// TIA Portal V17 export
// export: Created 2024-09-02T12:49:59.2213188Z, ExportSetting WithDefaults, DisplayName Totally Integrated Automation Portal, DisplayVersion V17, DisplayName TIA Portal Openness, DisplayVersion V17, DisplayName TIA Portal Version Control Interface, DisplayVersion V17, DisplayName STEP 7 Professional, DisplayVersion V17, DisplayName STEP 7 Safety, DisplayVersion V17, DisplayName WinCC Professional, DisplayVersion V17
DATA_BLOCK "LTLL_Data"   // DB556
TITLE = LTLL_Data
{ S7_Optimized_Access := 'TRUE'; DB_Accessible_From_OPC_UA := 'FALSE' }
AUTHOR : Siemens
FAMILY : HMI_Lite
NAME : LTLL_Data
VERSION : 8.10
// stored: AutoNumber true, DBAccessibleFromOPCUA false, IsOnlyStoredInLoadMemory false, IsRetainMemResEnabled false, IsWriteProtectedInAS false, MemoryReserve 100
   VAR RETAIN
      HMI { S7_SetPoint := 'True'} : Array[0..1] of "LTLL_typeData";
   END_VAR
BEGIN
   HMI[0..1]."version".high := 16#08;
   HMI[0..1]."version".middle := 16#01;
   HMI[0..1]."version".low := 16#00;
END_DATA_BLOCK
